FUNCTION_BLOCK ALPHA_LOOP
  {SET_ATTRIBUTE(OpcUa, SERVICE)}
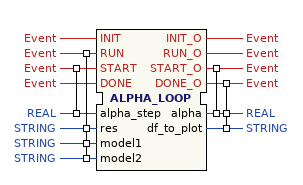
  EVENT_INPUT
    INIT;
    RUN WITH res, model1, model2; {SET_ATTRIBUTE(OpcUa, Method)}
    START WITH alpha_step; {SET_ATTRIBUTE(OpcUa, Method)}
    DONE; {SET_ATTRIBUTE(OpcUa, Method)}
  END_EVENT
  EVENT_OUTPUT
    INIT_O;
    RUN_O;
    START_O WITH alpha;
    DONE_O WITH alpha, df_to_plot;
  END_EVENT
  VAR_INPUT
    alpha_step : REAL; {SET_ATTRIBUTE(OpcUa, Variable.RUN)}
    res : STRING; {SET_ATTRIBUTE(OpcUa, Variable.RUN)}
    model1 : STRING; {SET_ATTRIBUTE(OpcUa, Variable.RUN)}
    model2 : STRING; {SET_ATTRIBUTE(OpcUa, Variable.RUN)}
  END_VAR
  VAR_OUTPUT
    alpha : REAL; {SET_ATTRIBUTE(OpcUa, Variable.RUN)}
    df_to_plot : STRING; {SET_ATTRIBUTE(OpcUa, Variable.RUN)}
  END_VAR
END_FUNCTION_BLOCK
